INTERFACE I_TIME_OF_DAY EXTENDS I_Datatype

PROPERTY PUBLIC Value : REFERENCE TO TIME_OF_DAY
GET
END_GET
END_PROPERTY

END_INTERFACE

(* stored: Version 1.1.0.1, ProductVersion 3.1.4024.15
   Itf I_TIME_OF_DAY: Id {c7e262db-2a91-00bc-1f03-ba314c220d34}
   Property Value: Id {810604ec-d4de-0fb7-36c6-311d484852ab}
   Get Get: Id {a6b506cc-0a96-0e23-1655-e70e7cbe6789} *)
